INTERFACE I_Log

METHOD AddLog : BOOL
VAR_INPUT
	sLog : STRING;
END_VAR
END_METHOD

END_INTERFACE

(* stored: Version 1.1.0.1, ProductVersion 3.1.4024.12
   Itf I_Log: Id {a2392562-2fbc-4d0c-b557-5145db6a7a8b}
   Method AddLog: Id {4a0597c3-5928-4193-911c-95bc632674c5} *)
